% RSLogix 500 project Simulated-Robotic-Pick-and-Place.RSS, saved by version 8.30.00.16 %
PROJECT "UNTITLED"    % processor: Bul.1763 MicroLogix 1100 Series B %

PROGRAM FILES
  LAD 2   6 rungs

DATA FILES
  O0 OUTPUT  4 elements
  I1 INPUT  6 elements
  S2 STATUS  66 elements
  B3 BINARY  1 elements
  T4 TIMER  3 elements
  C5 COUNTER  1 elements
  R6 CONTROL  1 elements
  N7 INTEGER  1 elements
  F8 FLOAT  1 elements

LADDER 2
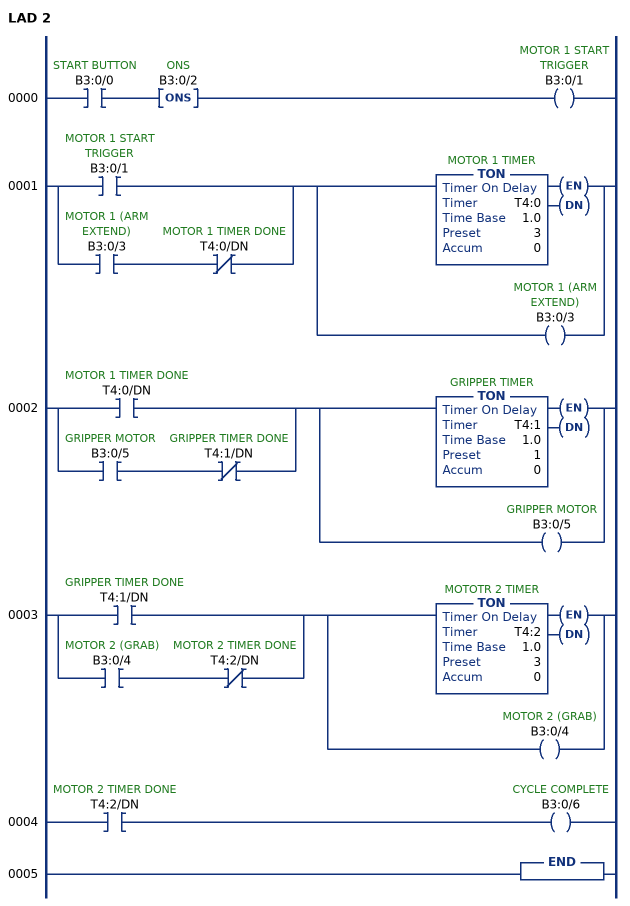
% Rung: 0 %
SOR XIC B3:0/0 ONS B3:0/2 OTE B3:0/1 EOR
%   B3:0/0  "START BUTTON" %
%   B3:0/2  "ONS" %
%   B3:0/1  "MOTOR 1 START TRIGGER" %
% Rung: 1 %
SOR BST XIC B3:0/1 NXB XIC B3:0/3 XIO T4:0/DN BND BST TON T4:0 1.0 3 0 NXB OTE B3:0/3 BND EOR
%   B3:0/1  "MOTOR 1 START TRIGGER" %
%   B3:0/3  "MOTOR 1 (ARM EXTEND)" %
%   T4:0/DN  "MOTOR 1 TIMER DONE" %
%   T4:0  "MOTOR 1 TIMER" %
% Rung: 2 %
SOR BST XIC T4:0/DN NXB XIC B3:0/5 XIO T4:1/DN BND BST TON T4:1 1.0 1 0 NXB OTE B3:0/5 BND EOR
%   T4:0/DN  "MOTOR 1 TIMER DONE" %
%   B3:0/5  "GRIPPER MOTOR" %
%   T4:1/DN  "GRIPPER TIMER DONE" %
%   T4:1  "GRIPPER TIMER" %
% Rung: 3 %
SOR BST XIC T4:1/DN NXB XIC B3:0/4 XIO T4:2/DN BND BST TON T4:2 1.0 3 0 NXB OTE B3:0/4 BND EOR
%   T4:1/DN  "GRIPPER TIMER DONE" %
%   B3:0/4  "MOTOR 2 (GRAB)" %
%   T4:2/DN  "MOTOR 2 TIMER DONE" %
%   T4:2  "MOTOTR 2 TIMER" %
% Rung: 4 %
SOR XIC T4:2/DN OTE B3:0/6 EOR
%   T4:2/DN  "MOTOR 2 TIMER DONE" %
%   B3:0/6  "CYCLE COMPLETE" %
% Rung: 5 %
SOR END EOR

DATA TABLE (non-zero values as saved)
DATA T4
% .PRE .ACC %
% T4:0 % 3 0
% T4:1 % 1 0
% T4:2 % 3 0
